FUNCTION_BLOCK FB_ActorStopRotateCommand IMPLEMENTS I_Command
VAR
	refFlyingHoist : REFERENCE TO FB_FlyingHoist;
END_VAR

METHOD Execute
IF (__ISVALIDREF(THIS^.refFlyingHoist)) THEN
	THIS^.refFlyingHoist.StopRotateCommand();
END_IF
END_METHOD

METHOD FB_init : BOOL
VAR_INPUT
	bInitRetains 	: BOOL; // if TRUE, the retain variables are initialized (warm start / cold start)
	bInCopyCode 	: BOOL;  // if TRUE, the instance afterwards gets moved into the copy code (online change)
	refFlyingHoist 	: REFERENCE TO FB_FlyingHoist;
END_VAR
IF (__ISVALIDREF(refFlyingHoist)) THEN
	THIS^.refFlyingHoist REF= refFlyingHoist;
ELSE
	THIS^.refFlyingHoist REF= 0;
END_IF
END_METHOD

END_FUNCTION_BLOCK

(* stored: Version 1.1.0.1, ProductVersion 3.1.4022.18
   POU FB_ActorStopRotateCommand: Id {d2d2c4a2-f534-4e61-b3d8-6964c09c6f2a}, SpecialFunc None
   Method Execute: Id {36115dc0-74e8-4d32-868a-6526c95a3359}
   Method FB_init: Id {7ba8bf25-e2d2-463a-a7ad-b1cb80d36bdc} *)
